// TwinCAT 3 PLC project PLC1
// ProgramVersion: 3.1.4022.7
// libraries:
//   Tc2_MC2, * (Beckhoff Automation GmbH)
//   Tc2_Standard, * (Beckhoff Automation GmbH)
//   Tc2_System, * (Beckhoff Automation GmbH)
//   Tc3_Module, * (Beckhoff Automation GmbH)
// project tree:
//   / ClassDiagram.TcCD (not stored), PlcTask.TcTTO
//   FBs/Commands/ FB_ActorDownCommand.TcPOU, FB_ShowOnCommnad.TcPOU, FB_ActorStopVerticalCommand.TcPOU, FB_ActorStopRotateCommand.TcPOU, FB_ActorRotateCCWCommand.TcPOU, FB_ActorRotateCWCommand.TcPOU, FB_ActorUpCommand.TcPOU, FB_FireShowModeCommand.TcPOU, FB_FirePyroModeCommand.TcPOU, FB_FireOffCommand.TcPOU, FB_MovingHeadOffCommand.TcPOU, FB_MovingHeadOnCommand.TcPOU
//   FBs/Invoker/ FB_ShowControlPanel.TcPOU
//   FBs/Receiver/ FB_FlameCannon.TcPOU, FB_FlyingHoist.TcPOU, FB_MovingHead.TcPOU
//   ITFs/Commands/ I_Command.TcIO
//   POUs/ MAIN.TcPOU
// real-time tasks:
//   TASK PlcTask: cycle T#10ms, priority 20, ADS port 350
// motion (NC):
//   TASK NC-Task 1 SAF: cycle T#2ms, priority 4, ADS port 501
//   TASK NC-Task 1 SVB: cycle T#10ms, priority 8, ADS port 511
//   AXIS FlyingHoist_Vert (id 1)
//     OtherSettings: AllowMotionCmdToSlave=true
//     encoder EncType=1
//     drive DrvType=5
//       Analog: ScaleFactorActTorque=0.1
//       TimeComp: TaskDelayCycles=1
//     controller CtrType=1
//       CtrPara: PriorControlFactor=1
//         Observer: BandWidth=20
//   AXIS FlyingHoist_Rot (id 2)
//     OtherSettings: AllowMotionCmdToSlave=true
//     encoder EncType=1
//     drive DrvType=5
//       Analog: ScaleFactorActTorque=0.1
//       TimeComp: TaskDelayCycles=1
//     controller CtrType=1
//       CtrPara: PriorControlFactor=1
//         Observer: BandWidth=20
// variable links:
//   PLC1/PLC1 Instance <-> NC-Task 1 SAF/Axes/FlyingHoist_Rot
//     PlcTask Inputs/MAIN.fbFlyingHoist.FlyingHoist_Rot.NcToPlc <-> Outputs/ToPlc
//     PlcTask Outputs/MAIN.fbFlyingHoist.FlyingHoist_Rot.PlcToNc <-> Inputs/FromPlc
//   PLC1/PLC1 Instance <-> NC-Task 1 SAF/Axes/FlyingHoist_Vert
//     PlcTask Inputs/MAIN.fbFlyingHoist.FlyingHoist_Vert.NcToPlc <-> Outputs/ToPlc
//     PlcTask Outputs/MAIN.fbFlyingHoist.FlyingHoist_Vert.PlcToNc <-> Inputs/FromPlc

CONFIGURATION PLC1
    RESOURCE PLC ON TwinCAT3
        TASK PlcTask(INTERVAL := T#10ms, PRIORITY := 20);
        PROGRAM MAIN WITH PlcTask : MAIN;
    END_RESOURCE
END_CONFIGURATION

// ---- ITFs/Commands/I_Command.TcIO
INTERFACE I_Command

METHOD Execute
END_METHOD

END_INTERFACE

// ---- POUs/MAIN.TcPOU
PROGRAM MAIN
VAR
	// Invoker
	fbHMI_panel				: FB_ShowControlPanel;
	fbPendant_panel			: FB_ShowControlPanel;
	
	// Receiver
	fbFlyingHoist			: FB_FlyingHoist;
	refFlyingHoist			: REFERENCE TO FB_FlyingHoist := fbFlyingHoist;	
	fbFlameCannon			: FB_FlameCannon;
	refFlameCannon			: REFERENCE TO FB_FlameCannon := fbFlameCannon;	
	fbMovingHead			: FB_MovingHead;
	refMovingHead			: REFERENCE TO FB_MovingHead := fbMovingHead;	

	// Commands
	fbActorDownCommand			: FB_ActorDownCommand(refFlyingHoist);
	fbActorUpCommand			: FB_ActorUpCommand(refFlyingHoist);
	fbActorRotateCCWCommand		: FB_ActorRotateCCWCommand(refFlyingHoist);
	fbActorRotateCWCommand		: FB_ActorRotateCWCommand(refFlyingHoist);
	fbActorStopRotateCommand	: FB_ActorStopRotateCommand(refFlyingHoist);
	fbActorStopVerticalCommand	: FB_ActorStopVerticalCommand(refFlyingHoist);
	fbFireShowModeCommand		: FB_FireShowModeCommand(fbFlameCannon);
	fbFirePyroModeCommand		: FB_FireShowModeCommand(fbFlameCannon);
	fbFireOffCommand			: FB_FireOffCommand(fbFlameCannon);
	fbMovingHeadOnCommand		: FB_MovingHeadOnCommand(fbMovingHead);
	fbMovingHeadOffCommand		: FB_MovingHeadOffCommand(fbMovingHead);
	fbShowOnCommnad				: FB_ShowOnCommnad(fbActorUpCommand, fbActorRotateCWCommand, fbFireShowModeCommand);
	bInit						: BOOL;
	
	fHoistVertPos				: LREAL;
	fHoistRotPos				: LREAL;
END_VAR

IF (NOT bInit) THEN
	fbHMI_panel.SetCommand(1, fbActorDownCommand);
	fbHMI_panel.SetCommand(2, fbActorUpCommand);
	fbHMI_panel.SetCommand(3, fbActorRotateCCWCommand);
	fbHMI_panel.SetCommand(4, fbActorRotateCWCommand);
	fbHMI_panel.SetCommand(5, fbActorStopVerticalCommand);
	fbHMI_panel.SetCommand(6, fbActorStopRotateCommand);
	fbHMI_panel.SetCommand(7, fbFireShowModeCommand);
	fbHMI_panel.SetCommand(8, fbFirePyroModeCommand);
	fbHMI_panel.SetCommand(9, fbFireOffCommand);
	fbHMI_panel.SetCommand(10, fbMovingHeadOnCommand);
	fbHMI_panel.SetCommand(11, fbMovingHeadOffCommand);
	fbHMI_panel.SetCommand(12, fbShowOnCommnad);
	
	fbPendant_panel.SetCommand(1, fbActorDownCommand);
	fbPendant_panel.SetCommand(2, fbActorUpCommand);
	fbPendant_panel.SetCommand(3, fbActorRotateCCWCommand);
	fbPendant_panel.SetCommand(4, fbActorRotateCWCommand);
	fbPendant_panel.SetCommand(5, fbActorStopVerticalCommand);
	fbPendant_panel.SetCommand(6, fbActorStopRotateCommand);

	
	bInit := TRUE;
ELSE
	fbHMI_panel();	
	fbPendant_panel();
END_IF


(* Trigger fbPendant_panel.arrSwitch[1 - 4] for moves, and arrSwitch[5 - 6] for stops.
OR
Trigger fbHMI_panel.arrSwitch[1 - 4] for moves, and arrSwitch[5 - 6] for stops. *)

// Check the positions of the hoist
fHoistRotPos 	:= fbFlyingHoist.RotationalPosition;
fHoistVertPos 	:= fbFlyingHoist.VerticalPosition;

END_PROGRAM

// ---- FBs/Invoker/FB_ShowControlPanel.TcPOU
FUNCTION_BLOCK FB_ShowControlPanel
VAR_INPUT
	arrSwitch		: ARRAY[1..C_MAXCOMMANDS] OF BOOL;
END_VAR
VAR
	aiCommand		: ARRAY[1..C_MAXCOMMANDS] OF I_Command;	
	arrRtrig		: ARRAY[1..C_MAXCOMMANDS] OF R_TRIG;
	nIndex			: INT;
END_VAR
VAR CONSTANT
	C_MAXCOMMANDS	: INT := 12;
END_VAR

FOR nIndex := 1 TO C_MAXCOMMANDS DO
	arrRtrig[nIndex](CLK := arrSwitch[nIndex]);
	IF aiCommand[nIndex] <> 0 THEN
		
		IF arrRtrig[nIndex].Q AND (aiCommand[nIndex] <> 0)THEN
				aiCommand[nIndex].Execute();	
		END_IF
				
	END_IF
END_FOR

METHOD FB_init : BOOL
VAR_INPUT
	bInitRetains : BOOL; // if TRUE, the retain variables are initialized (warm start / cold start)
	bInCopyCode : BOOL;  // if TRUE, the instance afterwards gets moved into the copy code (online change)
END_VAR
VAR
	nIndex : INT;
END_VAR
FOR nIndex := 1 TO C_MAXCOMMANDS DO
	aiCommand[nIndex] := 0;
END_FOR
END_METHOD

METHOD SetCommand : BOOL
VAR_INPUT
	nPosition		: INT;
	iCommand		: I_Command;
END_VAR
IF ((nPosition >= 1) AND (nPosition <= C_MAXCOMMANDS) AND (iCommand <> 0)) THEN
		THIS^.aiCommand[nPosition] := iCommand;
END_IF
END_METHOD

END_FUNCTION_BLOCK

// ---- FBs/Receiver/FB_FlyingHoist.TcPOU
FUNCTION_BLOCK FB_FlyingHoist
VAR
	FlyingHoist_Vert : Axis_Ref;
	FlyingHoist_Rot  : Axis_Ref;
	
	mcPower : ARRAY[1..2] OF MC_Power;
	mcJog	: ARRAY[1..2] OF MC_Jog;
	
	_RepIndexer : INT := 0;

END_VAR

METHOD ActorDown : BOOL
VAR_INPUT
END_VAR
_RepIndexer := 0;

REPEAT	
	mcJog[1](
		Axis:= FlyingHoist_Vert, 
		JogForward:= TRUE, 
		JogBackwards:= FALSE, 
		Velocity:= 500, 
		Acceleration:= 2000, 
		Deceleration:= 2000, 
		Jerk:=  2000);
	
	_RepIndexer := _RepIndexer + 1;
UNTIL
	_RepIndexer = 4
END_REPEAT
END_METHOD

METHOD ActorRotateCCW : BOOL
VAR_INPUT
END_VAR
_RepIndexer := 0;

REPEAT	
	mcJog[2](
		Axis:= FlyingHoist_Rot, 
		JogForward:= TRUE, 
		JogBackwards:= FALSE, 
		Velocity:= 500, 
		Acceleration:= 2000, 
		Deceleration:= 2000, 
		Jerk:=  2000);
		
	_RepIndexer := _RepIndexer + 1;
UNTIL
	_RepIndexer = 4
END_REPEAT
END_METHOD

METHOD ActorRotateCW : BOOL
VAR_INPUT
END_VAR
_RepIndexer := 0;

REPEAT	
	mcJog[2](
		Axis:= FlyingHoist_Rot, 
		JogForward:= FALSE, 
		JogBackwards:= TRUE, 
		Velocity:= 500, 
		Acceleration:= 2000, 
		Deceleration:= 2000, 
		Jerk:=  2000);
		
	_RepIndexer := _RepIndexer + 1;
UNTIL
	_RepIndexer = 4
END_REPEAT
END_METHOD

METHOD ActorUp : BOOL
VAR_INPUT
END_VAR
_RepIndexer := 0;

REPEAT	
	mcJog[1](
		Axis:= FlyingHoist_Vert, 
		JogForward:= FALSE, 
		JogBackwards:= TRUE, 
		Velocity:= 500, 
		Acceleration:= 2000, 
		Deceleration:= 2000, 
		Jerk:=  2000);
	
	_RepIndexer := _RepIndexer + 1;
UNTIL
	_RepIndexer = 4
END_REPEAT
END_METHOD

METHOD HoistEnable : BOOL
mcPower[1](
	Axis:= FlyingHoist_Vert, 
	Enable:= TRUE, 
	Enable_Positive:= TRUE, 
	Enable_Negative:= TRUE, 
	Override:= 100.00);
	
mcPower[2](
	Axis:= FlyingHoist_Rot, 
	Enable:= TRUE, 
	Enable_Positive:= TRUE, 
	Enable_Negative:= TRUE, 
	Override:= 100.00);
END_METHOD

PROPERTY RotationalPosition : LREAL
GET
RotationalPosition := THIS^.FlyingHoist_Rot.NcToPlc.ActPos;
END_GET
END_PROPERTY

METHOD StopRotateCommand : BOOL
_RepIndexer := 0;

REPEAT 
	mcJog[2](
		Axis:= FlyingHoist_Rot, 
		JogForward:= FALSE, 
		JogBackwards:= FALSE, 
		Velocity:= 500, 
		Acceleration:= 2000, 
		Deceleration:= 2000, 
		Jerk:=  2000);
		
	_RepIndexer := _RepIndexer + 1;
UNTIL
	_RepIndexer = 4
END_REPEAT
END_METHOD

METHOD StopVerticalCommand : BOOL
VAR_INPUT
END_VAR
_RepIndexer := 0;

REPEAT 

	mcJog[1](
		Axis:= FlyingHoist_Vert, 
		JogForward:= FALSE, 
		JogBackwards:= FALSE, 
		Velocity:= 500, 
		Acceleration:= 2000, 
		Deceleration:= 2000, 
		Jerk:=  2000);
		
			
	_RepIndexer := _RepIndexer + 1;
UNTIL
	_RepIndexer = 4
END_REPEAT
END_METHOD

PROPERTY VerticalPosition : LREAL
GET
VerticalPosition := THIS^.FlyingHoist_Vert.NcToPlc.ActPos;
END_GET
END_PROPERTY

END_FUNCTION_BLOCK

// ---- FBs/Receiver/FB_FlameCannon.TcPOU
FUNCTION_BLOCK FB_FlameCannon
VAR
	_Active : BOOL;
	_Level  : LREAL;
END_VAR

PROPERTY Active : BOOL
GET
Active := This^._Active;
END_GET
END_PROPERTY

PROPERTY Level : LREAL
GET
Level := This^._Level;
END_GET
END_PROPERTY

METHOD Off : BOOL
VAR_INPUT
END_VAR
This^._Active := FALSE;
END_METHOD

METHOD On : BOOL
VAR_INPUT
END_VAR
This^._Active := TRUE;
END_METHOD

METHOD SetLevel : BOOL
VAR_INPUT
	Level  : LREAL;
END_VAR
This^._Level := Level;
END_METHOD

END_FUNCTION_BLOCK

// ---- FBs/Receiver/FB_MovingHead.TcPOU
FUNCTION_BLOCK FB_MovingHead
VAR
	_Active : BOOL;
END_VAR

PROPERTY Active : BOOL
GET
Active := This^._Active;
END_GET
END_PROPERTY

METHOD Off : BOOL
VAR_INPUT
END_VAR
This^._Active := FALSE;
END_METHOD

METHOD On : BOOL
VAR_INPUT
END_VAR
This^._Active := TRUE;
END_METHOD

END_FUNCTION_BLOCK

// ---- FBs/Commands/FB_ActorDownCommand.TcPOU
FUNCTION_BLOCK FB_ActorDownCommand IMPLEMENTS I_Command
VAR
	refFlyingHoist : REFERENCE TO FB_FlyingHoist;
END_VAR

METHOD Execute
IF (__ISVALIDREF(THIS^.refFlyingHoist)) THEN
	THIS^.refFlyingHoist.HoistEnable();
	THIS^.refFlyingHoist.ActorDown();
END_IF
END_METHOD

METHOD FB_init : BOOL
VAR_INPUT
	bInitRetains 	: BOOL; // if TRUE, the retain variables are initialized (warm start / cold start)
	bInCopyCode 	: BOOL;  // if TRUE, the instance afterwards gets moved into the copy code (online change)
	refFlyingHoist 	: REFERENCE TO FB_FlyingHoist;
END_VAR
IF (__ISVALIDREF(refFlyingHoist)) THEN
	THIS^.refFlyingHoist REF= refFlyingHoist;
ELSE
	THIS^.refFlyingHoist REF= 0;
END_IF
END_METHOD

END_FUNCTION_BLOCK

// ---- FBs/Commands/FB_ActorUpCommand.TcPOU
FUNCTION_BLOCK FB_ActorUpCommand IMPLEMENTS I_Command
VAR
	refFlyingHoist : REFERENCE TO FB_FlyingHoist;
END_VAR

METHOD Execute
IF (__ISVALIDREF(THIS^.refFlyingHoist)) THEN
	THIS^.refFlyingHoist.HoistEnable();
	THIS^.refFlyingHoist.ActorUp();
END_IF
END_METHOD

METHOD FB_init : BOOL
VAR_INPUT
	bInitRetains 	: BOOL; // if TRUE, the retain variables are initialized (warm start / cold start)
	bInCopyCode 	: BOOL;  // if TRUE, the instance afterwards gets moved into the copy code (online change)
	refFlyingHoist 	: REFERENCE TO FB_FlyingHoist;
END_VAR
IF (__ISVALIDREF(refFlyingHoist)) THEN
	THIS^.refFlyingHoist REF= refFlyingHoist;
ELSE
	THIS^.refFlyingHoist REF= 0;
END_IF
END_METHOD

END_FUNCTION_BLOCK

// ---- FBs/Commands/FB_ActorRotateCCWCommand.TcPOU
FUNCTION_BLOCK FB_ActorRotateCCWCommand IMPLEMENTS I_Command
VAR
	refFlyingHoist : REFERENCE TO FB_FlyingHoist;
END_VAR

METHOD Execute
IF (__ISVALIDREF(THIS^.refFlyingHoist)) THEN
	THIS^.refFlyingHoist.HoistEnable();
	THIS^.refFlyingHoist.ActorRotateCCW();
END_IF
END_METHOD

METHOD FB_init : BOOL
VAR_INPUT
	bInitRetains 	: BOOL; // if TRUE, the retain variables are initialized (warm start / cold start)
	bInCopyCode 	: BOOL;  // if TRUE, the instance afterwards gets moved into the copy code (online change)
	refFlyingHoist 	: REFERENCE TO FB_FlyingHoist;
END_VAR
IF (__ISVALIDREF(refFlyingHoist)) THEN
	THIS^.refFlyingHoist REF= refFlyingHoist;
ELSE
	THIS^.refFlyingHoist REF= 0;
END_IF
END_METHOD

END_FUNCTION_BLOCK

// ---- FBs/Commands/FB_ActorRotateCWCommand.TcPOU
FUNCTION_BLOCK FB_ActorRotateCWCommand IMPLEMENTS I_Command
VAR
	refFlyingHoist : REFERENCE TO FB_FlyingHoist;
END_VAR

METHOD Execute
IF (__ISVALIDREF(THIS^.refFlyingHoist)) THEN
	THIS^.refFlyingHoist.HoistEnable();
	THIS^.refFlyingHoist.ActorRotateCW();
END_IF
END_METHOD

METHOD FB_init : BOOL
VAR_INPUT
	bInitRetains 	: BOOL; // if TRUE, the retain variables are initialized (warm start / cold start)
	bInCopyCode 	: BOOL;  // if TRUE, the instance afterwards gets moved into the copy code (online change)
	refFlyingHoist 	: REFERENCE TO FB_FlyingHoist;
END_VAR
IF (__ISVALIDREF(refFlyingHoist)) THEN
	THIS^.refFlyingHoist REF= refFlyingHoist;
ELSE
	THIS^.refFlyingHoist REF= 0;
END_IF
END_METHOD

END_FUNCTION_BLOCK

// ---- FBs/Commands/FB_ActorStopRotateCommand.TcPOU
FUNCTION_BLOCK FB_ActorStopRotateCommand IMPLEMENTS I_Command
VAR
	refFlyingHoist : REFERENCE TO FB_FlyingHoist;
END_VAR

METHOD Execute
IF (__ISVALIDREF(THIS^.refFlyingHoist)) THEN
	THIS^.refFlyingHoist.StopRotateCommand();
END_IF
END_METHOD

METHOD FB_init : BOOL
VAR_INPUT
	bInitRetains 	: BOOL; // if TRUE, the retain variables are initialized (warm start / cold start)
	bInCopyCode 	: BOOL;  // if TRUE, the instance afterwards gets moved into the copy code (online change)
	refFlyingHoist 	: REFERENCE TO FB_FlyingHoist;
END_VAR
IF (__ISVALIDREF(refFlyingHoist)) THEN
	THIS^.refFlyingHoist REF= refFlyingHoist;
ELSE
	THIS^.refFlyingHoist REF= 0;
END_IF
END_METHOD

END_FUNCTION_BLOCK

// ---- FBs/Commands/FB_ActorStopVerticalCommand.TcPOU
FUNCTION_BLOCK FB_ActorStopVerticalCommand IMPLEMENTS I_Command
VAR
	refFlyingHoist : REFERENCE TO FB_FlyingHoist;
END_VAR

METHOD Execute
IF (__ISVALIDREF(THIS^.refFlyingHoist)) THEN
	THIS^.refFlyingHoist.StopVerticalCommand();
END_IF
END_METHOD

METHOD FB_init : BOOL
VAR_INPUT
	bInitRetains 	: BOOL; // if TRUE, the retain variables are initialized (warm start / cold start)
	bInCopyCode 	: BOOL;  // if TRUE, the instance afterwards gets moved into the copy code (online change)
	refFlyingHoist 	: REFERENCE TO FB_FlyingHoist;
END_VAR
IF (__ISVALIDREF(refFlyingHoist)) THEN
	THIS^.refFlyingHoist REF= refFlyingHoist;
ELSE
	THIS^.refFlyingHoist REF= 0;
END_IF
END_METHOD

END_FUNCTION_BLOCK

// ---- FBs/Commands/FB_FireShowModeCommand.TcPOU
FUNCTION_BLOCK FB_FireShowModeCommand IMPLEMENTS I_Command
VAR
	refFlameCannon : REFERENCE TO FB_FlameCannon;
END_VAR

METHOD Execute
IF (__ISVALIDREF(THIS^.refFlameCannon)) THEN
	THIS^.refFlameCannon.On();
	THIS^.refFlameCannon.SetLevel(25.50);
END_IF
END_METHOD

METHOD FB_init : BOOL
VAR_INPUT
	bInitRetains 	: BOOL; // if TRUE, the retain variables are initialized (warm start / cold start)
	bInCopyCode 	: BOOL;  // if TRUE, the instance afterwards gets moved into the copy code (online change)
	refFlameCannon 	: REFERENCE TO FB_FlameCannon;
END_VAR
IF (__ISVALIDREF(refFlameCannon)) THEN
	THIS^.refFlameCannon REF= refFlameCannon;
ELSE
	THIS^.refFlameCannon REF= 0;
END_IF
END_METHOD

END_FUNCTION_BLOCK

// ---- FBs/Commands/FB_FireOffCommand.TcPOU
FUNCTION_BLOCK FB_FireOffCommand IMPLEMENTS I_Command
VAR
	refFlameCannon : REFERENCE TO FB_FlameCannon;
END_VAR

METHOD Execute
IF (__ISVALIDREF(THIS^.refFlameCannon)) THEN
	THIS^.refFlameCannon.Off();
END_IF
END_METHOD

METHOD FB_init : BOOL
VAR_INPUT
	bInitRetains 	: BOOL; // if TRUE, the retain variables are initialized (warm start / cold start)
	bInCopyCode 	: BOOL;  // if TRUE, the instance afterwards gets moved into the copy code (online change)
	refFlameCannon 	: REFERENCE TO FB_FlameCannon;
END_VAR
IF (__ISVALIDREF(refFlameCannon)) THEN
	THIS^.refFlameCannon REF= refFlameCannon;
ELSE
	THIS^.refFlameCannon REF= 0;
END_IF
END_METHOD

END_FUNCTION_BLOCK

// ---- FBs/Commands/FB_MovingHeadOnCommand.TcPOU
FUNCTION_BLOCK FB_MovingHeadOnCommand IMPLEMENTS I_Command
VAR
	refMovingHead : REFERENCE TO FB_MovingHead;
END_VAR

METHOD Execute
IF (__ISVALIDREF(THIS^.refMovingHead)) THEN
	THIS^.refMovingHead.On();
END_IF
END_METHOD

METHOD FB_init : BOOL
VAR_INPUT
	bInitRetains 	: BOOL; // if TRUE, the retain variables are initialized (warm start / cold start)
	bInCopyCode 	: BOOL;  // if TRUE, the instance afterwards gets moved into the copy code (online change)
	refMovingHead 	: REFERENCE TO FB_MovingHead;
END_VAR
IF (__ISVALIDREF(refMovingHead)) THEN
	THIS^.refMovingHead REF= refMovingHead;
ELSE
	THIS^.refMovingHead REF= 0;
END_IF
END_METHOD

END_FUNCTION_BLOCK

// ---- FBs/Commands/FB_MovingHeadOffCommand.TcPOU
FUNCTION_BLOCK FB_MovingHeadOffCommand IMPLEMENTS I_Command
VAR
	refMovingHead : REFERENCE TO FB_MovingHead;
END_VAR

METHOD Execute
IF (__ISVALIDREF(THIS^.refMovingHead)) THEN
	THIS^.refMovingHead.Off();
END_IF
END_METHOD

METHOD FB_init : BOOL
VAR_INPUT
	bInitRetains 	: BOOL; // if TRUE, the retain variables are initialized (warm start / cold start)
	bInCopyCode 	: BOOL;  // if TRUE, the instance afterwards gets moved into the copy code (online change)
	refMovingHead 	: REFERENCE TO FB_MovingHead;
END_VAR
IF (__ISVALIDREF(refMovingHead)) THEN
	THIS^.refMovingHead REF= refMovingHead;
ELSE
	THIS^.refMovingHead REF= 0;
END_IF
END_METHOD

END_FUNCTION_BLOCK

// ---- FBs/Commands/FB_ShowOnCommnad.TcPOU
FUNCTION_BLOCK FB_ShowOnCommnad IMPLEMENTS I_Command
VAR
	aiCommand : ARRAY[1..3] OF I_Command;
END_VAR

METHOD Execute
VAR
	nIndex		: INT;
END_VAR
FOR nIndex := 1 TO 3 DO
	IF (THIS^.aiCommand[nIndex] <> 0) THEN
		THIS^.aiCommand[nIndex].Execute();
	END_IF
END_FOR
END_METHOD

METHOD FB_init : BOOL
VAR_INPUT
	bInitRetains 	: BOOL; // if TRUE, the retain variables are initialized (warm start / cold start)
	bInCopyCode 	: BOOL;  // if TRUE, the instance afterwards gets moved into the copy code (online change)
	iCommand01 : I_Command;
	iCommand02 : I_Command;
	iCommand03 : I_Command;
END_VAR
THIS^.aiCommand[1] := 0;
THIS^.aiCommand[2] := 0;
THIS^.aiCommand[3] := 0;

IF (iCommand01 <> 0) THEN
	THIS^.aiCommand[1] := iCommand01;
END_IF
IF (iCommand02 <> 0) THEN
	THIS^.aiCommand[2] := iCommand02;
END_IF
IF (iCommand03 <> 0) THEN
	THIS^.aiCommand[3] := iCommand03;
END_IF
END_METHOD

END_FUNCTION_BLOCK

// ---- FBs/Commands/FB_FirePyroModeCommand.TcPOU
FUNCTION_BLOCK FB_FirePyroModeCommand IMPLEMENTS I_Command
VAR
	refFlameCannon : REFERENCE TO FB_FlameCannon;
END_VAR

METHOD Execute
IF (__ISVALIDREF(THIS^.refFlameCannon)) THEN
	THIS^.refFlameCannon.On();
	THIS^.refFlameCannon.SetLevel(95.00);
END_IF
END_METHOD

METHOD FB_init : BOOL
VAR_INPUT
	bInitRetains 	: BOOL; // if TRUE, the retain variables are initialized (warm start / cold start)
	bInCopyCode 	: BOOL;  // if TRUE, the instance afterwards gets moved into the copy code (online change)
	refFlameCannon 	: REFERENCE TO FB_FlameCannon;
END_VAR
IF (__ISVALIDREF(refFlameCannon)) THEN
	THIS^.refFlameCannon REF= refFlameCannon;
ELSE
	THIS^.refFlameCannon REF= 0;
END_IF
END_METHOD

END_FUNCTION_BLOCK
